# EPICS substitutions: icefrdgeSup/proportional_valve.substitutions
file proportional_valve.template {
  pattern
    {P, PORT, VALVE_NUM, IF_ONE}

    {"\$(P)", "\$(PORT)", "1", ""}
    {"\$(P)", "\$(PORT)", "2", "#"}
    {"\$(P)", "\$(PORT)", "4", "#"}
}
